Staubli VAL3: onEnterEvent.pgx

program onEnterEvent()
begin
  //
  // NB sEvent is the selected
  // element in the LIST
  //
  //
  // Change the cycle to do
  //
  if sEvent!=""
    call changeCycle(nIndex,sEvent)
    // logMsg
    logMsg("[KERNEL] CYCLEKEYEVENT:Change cycle to do for the program: "+sEvent+" at position: "+toString("",nIndex))
  endIf
end
